Staubli VAL3: refreshPoints.pgx

program refreshPoints(Trajectory& x_tTraj[])
  local num i
  local num l_nSize
  local string l_sEvent
  local string l_sItem
  local num j
  local num l_nIndex
  local string l_sData
  local string l_sType
begin
  // create the list
  call usePoint:type(21,0,x_tTraj.sID)
  // get the size
  call usePoint:listempty()
  l_nSize=size(x_tTraj.tSuper)
  for i=0 to l_nSize-1
    // add..
    l_sEvent=x_tTraj.tSuper[i].comment
    l_sItem=toString("2",i+1)+" "+l_sEvent
    nPointLine[i]=l_nIndex
    call usePoint:listadd(l_sItem)
    l_nIndex=l_nIndex+1
    if saveData:bShowItem
      // search for tCP ON OFF
      if x_tTraj.tSuper[i].nTcpAction==1
        l_sItem="  -TCP ON"
      elseIf x_tTraj.tSuper[i].nTcpAction==2
        l_sItem="  -TCP OFF"
      endIf
      if x_tTraj.tSuper[i].nTcpAction>0
        call usePoint:listadd(l_sItem)
        l_nIndex=l_nIndex+1
      endIf
      // scan the action...
      for j=0 to size(x_tTraj.tSuper[i].iInstr)-1
        if x_tTraj.tSuper[i].iInstr[j].sType!=""
          l_sData=x_tTraj.tSuper[i].iInstr[j].sData
          l_sType=x_tTraj.tSuper[i].iInstr[j].sType
          call saveInputOutput:replaceIO(l_sData,l_sType,l_sData)
          l_sItem=l_sType+" "+l_sData
          l_sItem="  -"+l_sItem
          call usePoint:listadd(l_sItem)
          l_nIndex=l_nIndex+1
        endIf
      endFor
    endIf
  endFor
end
